PROGRAM PRG_DIAGNOSTIC
VAR
   fbTime : FB_LocalSystemTime := ( bEnable := TRUE, dwCycle := 1 );
   logTimer : TON := ( IN := TRUE, PT := T#1000ms );

   plcName : STRING[15];

   {attribute 'pytmc' := ' pv: simHeartbeat '}
   simHeartbeat AT %I* : UINT := 0;
   {attribute 'pytmc' := ' pv: plcHeartbeat '}
   plcHeartbeat : UDINT := 0;
   {attribute 'pytmc' := ' pv: plcInfo '}
   plcInfo : STRING[40];
   {attribute 'pytmc' := ' pv: plcLocalTime '}
   plcLocalTime : STRING[25];
   
END_VAR

plcHeartbeat := plcHeartbeat + 1;
IF plcHeartbeat > 4294967000
   THEN plcHeartbeat := 0;
END_IF

// get timestamp as string every second
fbTime();
logTimer( IN := fbTime.bValid );
IF logTimer.Q THEN
   logTimer( IN := FALSE ); logTimer( IN := fbTime.bValid );
   plcLocalTime := SYSTEMTIME_TO_STRING(fbTime.systemTime);
END_IF

// make an info string
plcName := 'Prototype PLC: ';
plcInfo := CONCAT(plcName, plcLocalTime);

END_PROGRAM

(* stored: Version 1.1.0.1, ProductVersion 3.1.4022.18
   POU PRG_DIAGNOSTIC: Id {d6e7a1ee-1aeb-429b-a7e8-4b912c0cf7c2}, SpecialFunc None *)
